// TIA Portal V17 export
// export: Created 2024-06-14T09:53:03.8054565Z, ExportSetting WithDefaults, DisplayName Totally Integrated Automation Portal, DisplayVersion V17, DisplayName TIA Portal Openness, DisplayVersion V17, DisplayName TIA Portal Version Control Interface, DisplayVersion V17, DisplayName Simotion SCOUT TIA, DisplayVersion 5.4.3.0, DisplayName SINAMICS Startdrive Advanced, DisplayVersion V17 SP1 Update 1, DisplayName SINAMICS Startdrive G110M, G120, G120C, G120D, G120P, G115D, DisplayVersion V17 SP1 Update 1, DisplayName SINAMICS Startdrive G130, G150, S120, S150, SINAMICS MV, S210, DisplayVersion V17 SP1 Update 1, DisplayName STEP 7 Professional, DisplayVersion V17, DisplayName STEP 7 Safety, DisplayVersion V17, DisplayName WinCC Professional, DisplayVersion V17
DATA_BLOCK "hmi"   // DB27
{ S7_Optimized_Access := 'TRUE' }
VERSION : 0.1
// stored: AutoNumber true, DBAccessibleFromOPCUA true, IsOnlyStoredInLoadMemory false, IsRetainMemResEnabled false, IsWriteProtectedInAS false, MemoryReserve 100
   VAR
      Start : Bool;
      Actual_Weight_cylinder : Real;
      Production_Count : Int;
      Pervious_Day_Count : Int;
      "Cylinder _rejected_S1" : Int;
      Cylinder_Rejected_S6 : Int;
      Truck_No : String;
      Dealer_Code : String;
      Total_Cylinder_Count : Int := 1;
      Domestic_Cylinder_Count : Int;
      Commercial_Cylinder_Count : Int;
      Reset : Bool;
      Cylinder_Count_Actual : Real;
      "Load S1" : Bool;
      "Load S2" : Bool;
      "Load S3" : Bool;
      "Load S4" : Bool;
      "Load S5" : Bool;
      "Load S46" : Bool;
      "Load S56" : Bool;
      "Load S68" : Bool;
      "Load S67" : Bool;
      "Load S78" : Bool;
      Buffer_Reinitialize : Bool;
      cy_t1 : String;
      cy_t2 : String;
      cy_t3 : String;
      cy_t4 : String;
      cy_t5 : String;
      BPCL : Bool;
      MALABAR : Bool;
      In_range : Int;
      "sensing time" : Int;
      password : Int;
      "tare check" : Bool;
      "tare check_1" : Bool;
      "data count" : Int;
      "Load S35" : Bool;
      "Load S56_L2" : Bool;
      "tare check_2" : Bool;
   END_VAR
   VAR RETAIN
      "AUTO/MAN_L1" : Bool;
      "AUTO/MAN_L2" : Bool;
   END_VAR
   VAR
      DIVERTER : Bool;
      NO_itmes_tocopy : Int;
   END_VAR
BEGIN
END_DATA_BLOCK
